(* IEC 61131-3 sources: teller/JD_Teller_LC2_V11/Class/Box_Editer (part 2) *)

            //3-punt 2300
            elsif i = 2 then

                  DoosData^.MinMax[i].T_Max := 2000;
                  DoosData^.MinMax[i].T_Min := 160;
                  DoosData^.MinMax[i].U_Max := 300;
                  DoosData^.MinMax[i].U_Min := 50;
                  DoosData^.MinMax[i].V_Max := 300;
                  DoosData^.MinMax[i].V_Min := 50;
                  DoosData^.MinMax[i].W_Max := 2300;
                  DoosData^.MinMax[i].W_Min := 510;
                  DoosData^.MinMax[i].X_Max := 820;
                  DoosData^.MinMax[i].X_Min := 50;
                  DoosData^.MinMax[i].Y_Max := 820;
                  DoosData^.MinMax[i].Y_Min := 150;
                  DoosData^.MinMax[i].Z_Max := 300;
                  DoosData^.MinMax[i].Z_Min := 0;
                  DoosData^.MinMax[i].Offset_Max := 1150;
                  DoosData^.MinMax[i].Offset_Min := 0;

            //3-punt vakverdeling 2300
            elsif i = 3 then

                  DoosData^.MinMax[i].T_Max := 2000;
                  DoosData^.MinMax[i].T_Min := 320;
                  DoosData^.MinMax[i].U_Max := 300;
                  DoosData^.MinMax[i].U_Min := 30;
                  DoosData^.MinMax[i].V_Max := 300;
                  DoosData^.MinMax[i].V_Min := 30;
                  DoosData^.MinMax[i].W_Max := 1900;
                  DoosData^.MinMax[i].W_Min := 500;
                  DoosData^.MinMax[i].X_Max := 820;
                  DoosData^.MinMax[i].X_Min := 150;
                  DoosData^.MinMax[i].Y_Max := 820;
                  DoosData^.MinMax[i].Y_Min := 100;
                  DoosData^.MinMax[i].Z_Max := 300;
                  DoosData^.MinMax[i].Z_Min := 0;
                  DoosData^.MinMax[i].Offset_Max := 1150;
                  DoosData^.MinMax[i].Offset_Min := 0;

            //4-punt infold 2300
            elsif i = 4 then

                  DoosData^.MinMax[i].T_Max := 2000;
                  DoosData^.MinMax[i].T_Min := 150;
                  DoosData^.MinMax[i].U_Max := 300;
                  DoosData^.MinMax[i].U_Min := 30;
                  DoosData^.MinMax[i].V_Max := 300;
                  DoosData^.MinMax[i].V_Min := 30;
                  DoosData^.MinMax[i].W_Max := 0;
                  DoosData^.MinMax[i].W_Min := 0;
                  DoosData^.MinMax[i].X_Max := 300;
                  DoosData^.MinMax[i].X_Min := 30;
                  DoosData^.MinMax[i].Y_Max := 1480;
                  DoosData^.MinMax[i].Y_Min := 250;
                  DoosData^.MinMax[i].Z_Max := 300;
                  DoosData^.MinMax[i].Z_Min := 0;
                  DoosData^.MinMax[i].Offset_Max := 1150;
                  DoosData^.MinMax[i].Offset_Min := 0;

            //4-punt outfold 2300
            elsif i = 5 then

                  DoosData^.MinMax[i].T_Max := 2000;
                  DoosData^.MinMax[i].T_Min := 150;
                  DoosData^.MinMax[i].U_Max := 300;
                  DoosData^.MinMax[i].U_Min := 30;
                  DoosData^.MinMax[i].V_Max := 300;
                  DoosData^.MinMax[i].V_Min := 30;
                  DoosData^.MinMax[i].W_Max := 0;
                  DoosData^.MinMax[i].W_Min := 0;
                  DoosData^.MinMax[i].X_Max := 300;
                  DoosData^.MinMax[i].X_Min := 30;
                  DoosData^.MinMax[i].Y_Max := 1180;
                  DoosData^.MinMax[i].Y_Min := 250;
                  DoosData^.MinMax[i].Z_Max := 300;
                  DoosData^.MinMax[i].Z_Min := 0;
                  DoosData^.MinMax[i].Offset_Max := 1150;
                  DoosData^.MinMax[i].Offset_Min := 0;

            //4-punt met deksel 2300
            elsif i = 6 then

                  DoosData^.MinMax[i].T_Max := 2000;
                  DoosData^.MinMax[i].T_Min := 150;
                  DoosData^.MinMax[i].U_Max := 300;
                  DoosData^.MinMax[i].U_Min := 30;
                  DoosData^.MinMax[i].V_Max := 300;
                  DoosData^.MinMax[i].V_Min := 30;
                  DoosData^.MinMax[i].W_Max := 2170;
                  DoosData^.MinMax[i].W_Min := 0;
                  DoosData^.MinMax[i].X_Max := 300;
                  DoosData^.MinMax[i].X_Min := 30;
                  DoosData^.MinMax[i].Y_Max := 1480;
                  DoosData^.MinMax[i].Y_Min := 250;
                  DoosData^.MinMax[i].Z_Max := 300;
                  DoosData^.MinMax[i].Z_Min := 0;
                  DoosData^.MinMax[i].Offset_Max := 1150;
                  DoosData^.MinMax[i].Offset_Min := 0;

            //4-punt dubbele wand 2300
            elsif i = 7 then

                  DoosData^.MinMax[i].T_Max := 2000;
                  DoosData^.MinMax[i].T_Min := 150;
                  DoosData^.MinMax[i].U_Max := 300;
                  DoosData^.MinMax[i].U_Min := 30;
                  DoosData^.MinMax[i].V_Max := 300;
                  DoosData^.MinMax[i].V_Min := 30;
                  DoosData^.MinMax[i].W_Max := 2170;
                  DoosData^.MinMax[i].W_Min := 0;
                  DoosData^.MinMax[i].X_Max := 300;
                  DoosData^.MinMax[i].X_Min := 30;
                  DoosData^.MinMax[i].Y_Max := 1480;
                  DoosData^.MinMax[i].Y_Min := 250;
                  DoosData^.MinMax[i].Z_Max := 300;
                  DoosData^.MinMax[i].Z_Min := 0;
                  DoosData^.MinMax[i].Offset_Max := 1150;
                  DoosData^.MinMax[i].Offset_Min := 0;

            //6-punt in/in 2300
            elsif i = 8 then

                  DoosData^.MinMax[i].T_Max := 2000;
                  DoosData^.MinMax[i].T_Min := 150;
                  DoosData^.MinMax[i].U_Max := 300;
                  DoosData^.MinMax[i].U_Min := 30;
                  DoosData^.MinMax[i].V_Max := 300;
                  DoosData^.MinMax[i].V_Min := 30;
                  DoosData^.MinMax[i].W_Max := 2170;
                  DoosData^.MinMax[i].W_Min := 0;
                  DoosData^.MinMax[i].X_Max := 300;
                  DoosData^.MinMax[i].X_Min := 30;
                  DoosData^.MinMax[i].Y_Max := 1480;
                  DoosData^.MinMax[i].Y_Min := 250;
                  DoosData^.MinMax[i].Z_Max := 300;
                  DoosData^.MinMax[i].Z_Min := 0;
                  DoosData^.MinMax[i].Offset_Max := 1150;
                  DoosData^.MinMax[i].Offset_Min := 0;

            //6-punt in/out 2300
            elsif i = 9 then

                  DoosData^.MinMax[i].T_Max := 2000;
                  DoosData^.MinMax[i].T_Min := 150;
                  DoosData^.MinMax[i].U_Max := 300;
                  DoosData^.MinMax[i].U_Min := 30;
                  DoosData^.MinMax[i].V_Max := 300;
                  DoosData^.MinMax[i].V_Min := 30;
                  DoosData^.MinMax[i].W_Max := 2170;
                  DoosData^.MinMax[i].W_Min := 0;
                  DoosData^.MinMax[i].X_Max := 300;
                  DoosData^.MinMax[i].X_Min := 30;
                  DoosData^.MinMax[i].Y_Max := 1480;
                  DoosData^.MinMax[i].Y_Min := 250;
                  DoosData^.MinMax[i].Z_Max := 300;
                  DoosData^.MinMax[i].Z_Min := 0;
                  DoosData^.MinMax[i].Offset_Max := 1150;
                  DoosData^.MinMax[i].Offset_Min := 0;

            //6-punt in/in 2300
            elsif i = 10 then

                  DoosData^.MinMax[i].T_Max := 2000;
                  DoosData^.MinMax[i].T_Min := 150;
                  DoosData^.MinMax[i].U_Max := 300;
                  DoosData^.MinMax[i].U_Min := 30;
                  DoosData^.MinMax[i].V_Max := 300;
                  DoosData^.MinMax[i].V_Min := 30;
                  DoosData^.MinMax[i].W_Max := 2170;
                  DoosData^.MinMax[i].W_Min := 0;
                  DoosData^.MinMax[i].X_Max := 300;
                  DoosData^.MinMax[i].X_Min := 30;
                  DoosData^.MinMax[i].Y_Max := 1480;
                  DoosData^.MinMax[i].Y_Min := 250;
                  DoosData^.MinMax[i].Z_Max := 300;
                  DoosData^.MinMax[i].Z_Min := 0;
                  DoosData^.MinMax[i].Offset_Max := 1150;
                  DoosData^.MinMax[i].Offset_Min := 0;

            //3-punt (gespiegeld) 2300
            elsif i = 11 then

                  DoosData^.MinMax[i].T_Max := 2000;
                  DoosData^.MinMax[i].T_Min := 160;
                  DoosData^.MinMax[i].U_Max := 300;
                  DoosData^.MinMax[i].U_Min := 50;
                  DoosData^.MinMax[i].V_Max := 300;
                  DoosData^.MinMax[i].V_Min := 50;
                  DoosData^.MinMax[i].W_Max := 2300;
                  DoosData^.MinMax[i].W_Min := 510;
                  DoosData^.MinMax[i].X_Max := 820;
                  DoosData^.MinMax[i].X_Min := 50;
                  DoosData^.MinMax[i].Y_Max := 820;
                  DoosData^.MinMax[i].Y_Min := 150;
                  DoosData^.MinMax[i].Z_Max := 300;
                  DoosData^.MinMax[i].Z_Min := 0;
                  DoosData^.MinMax[i].Offset_Max := 1150;
                  DoosData^.MinMax[i].Offset_Min := 0;

            //3-punt (Storaenzo Jonkoping) 2300
            elsif i = 12 then

                  DoosData^.MinMax[i].T_Max := 2000;
                  DoosData^.MinMax[i].T_Min := 160;
                  DoosData^.MinMax[i].U_Max := 300;
                  DoosData^.MinMax[i].U_Min := 50;
                  DoosData^.MinMax[i].V_Max := 300;
                  DoosData^.MinMax[i].V_Min := 50;
                  DoosData^.MinMax[i].W_Max := 2300;
                  DoosData^.MinMax[i].W_Min := 510;
                  DoosData^.MinMax[i].X_Max := 820;
                  DoosData^.MinMax[i].X_Min := 50;
                  DoosData^.MinMax[i].Y_Max := 820;
                  DoosData^.MinMax[i].Y_Min := 150;
                  DoosData^.MinMax[i].Z_Max := 300;
                  DoosData^.MinMax[i].Z_Min := 0;
                  DoosData^.MinMax[i].Offset_Max := 1150;
                  DoosData^.MinMax[i].Offset_Min := 0;

            //langsnaad2 2300
            elsif i = 13 then

                  DoosData^.MinMax[i].T_Max := 2000;
                  DoosData^.MinMax[i].T_Min := 160;
                  DoosData^.MinMax[i].U_Max := 300;
                  DoosData^.MinMax[i].U_Min := 50;
                  DoosData^.MinMax[i].V_Max := 300;
                  DoosData^.MinMax[i].V_Min := 50;
                  DoosData^.MinMax[i].W_Max := 2300;
                  DoosData^.MinMax[i].W_Min := 510;
                  DoosData^.MinMax[i].X_Max := 820;
                  DoosData^.MinMax[i].X_Min := 50;
                  DoosData^.MinMax[i].Y_Max := 820;
                  DoosData^.MinMax[i].Y_Min := 150;
                  DoosData^.MinMax[i].Z_Max := 300;
                  DoosData^.MinMax[i].Z_Min := 0;
                  DoosData^.MinMax[i].Offset_Max := 1150;
                  DoosData^.MinMax[i].Offset_Min := 0;

            //3-punt2 2300
            elsif i = 14 then

                  DoosData^.MinMax[i].T_Max := 2000;
                  DoosData^.MinMax[i].T_Min := 160;
                  DoosData^.MinMax[i].U_Max := 300;
                  DoosData^.MinMax[i].U_Min := 50;
                  DoosData^.MinMax[i].V_Max := 300;
                  DoosData^.MinMax[i].V_Min := 50;
                  DoosData^.MinMax[i].W_Max := 2300;
                  DoosData^.MinMax[i].W_Min := 510;
                  DoosData^.MinMax[i].X_Max := 820;
                  DoosData^.MinMax[i].X_Min := 50;
                  DoosData^.MinMax[i].Y_Max := 820;
                  DoosData^.MinMax[i].Y_Min := 150;
                  DoosData^.MinMax[i].Z_Max := 300;
                  DoosData^.MinMax[i].Z_Min := 0;
                  DoosData^.MinMax[i].Offset_Max := 1150;
                  DoosData^.MinMax[i].Offset_Min := 0;
          end_if;
        end_for;
  end_if;

  if    Presets_MinMax =  m2800 then

        for i:= 1 to 14 do

            DoosData^.MinMax[i].Max_Invoer_Lengte  := 2000;
            DoosData^.MinMax[i].Max_Invoer_Breedte := 2800;

              //langsnaad 2800
            if    i = 1 then

                  DoosData^.MinMax[i].T_Max := 2000;
                  DoosData^.MinMax[i].T_Min := 160;
                  DoosData^.MinMax[i].U_Max := 300;
                  DoosData^.MinMax[i].U_Min := 80;
                  DoosData^.MinMax[i].V_Max := 0;
                  DoosData^.MinMax[i].V_Min := 0;
                  DoosData^.MinMax[i].W_Max := 2800;
                  DoosData^.MinMax[i].W_Min := 510;
                  DoosData^.MinMax[i].X_Max := 1000;
                  DoosData^.MinMax[i].X_Min := 80;
                  DoosData^.MinMax[i].Y_Max := 1000;
                  DoosData^.MinMax[i].Y_Min := 150;
                  DoosData^.MinMax[i].Z_Max := 300;
                  DoosData^.MinMax[i].Z_Min := 0;
                  DoosData^.MinMax[i].Offset_Max := 1400;
                  DoosData^.MinMax[i].Offset_Min := 0;

            //3-punt 2800
            elsif i = 2 then

                  DoosData^.MinMax[i].T_Max := 2000;
                  DoosData^.MinMax[i].T_Min := 160;
                  DoosData^.MinMax[i].U_Max := 300;
                  DoosData^.MinMax[i].U_Min := 80;
                  DoosData^.MinMax[i].V_Max := 300;
                  DoosData^.MinMax[i].V_Min := 80;
                  DoosData^.MinMax[i].W_Max := 2800;
                  DoosData^.MinMax[i].W_Min := 510;
                  DoosData^.MinMax[i].X_Max := 1000;
                  DoosData^.MinMax[i].X_Min := 80;
                  DoosData^.MinMax[i].Y_Max := 1000;
                  DoosData^.MinMax[i].Y_Min := 150;
                  DoosData^.MinMax[i].Z_Max := 300;
                  DoosData^.MinMax[i].Z_Min := 0;
                  DoosData^.MinMax[i].Offset_Max := 1400;
                  DoosData^.MinMax[i].Offset_Min := 0;

            //3-punt vakverdeling 2800
            elsif i = 3 then

                  DoosData^.MinMax[i].T_Max := 2000;
                  DoosData^.MinMax[i].T_Min := 320;
                  DoosData^.MinMax[i].U_Max := 300;
                  DoosData^.MinMax[i].U_Min := 30;
                  DoosData^.MinMax[i].V_Max := 300;
                  DoosData^.MinMax[i].V_Min := 30;
                  DoosData^.MinMax[i].W_Max := 2400;
                  DoosData^.MinMax[i].W_Min := 500;
                  DoosData^.MinMax[i].X_Max := 1000;
                  DoosData^.MinMax[i].X_Min := 150;
                  DoosData^.MinMax[i].Y_Max := 1000;
                  DoosData^.MinMax[i].Y_Min := 100;
                  DoosData^.MinMax[i].Z_Max := 300;
                  DoosData^.MinMax[i].Z_Min := 0;
                  DoosData^.MinMax[i].Offset_Max := 1150;
                  DoosData^.MinMax[i].Offset_Min := 0;

            //4-punt infold 2800
            elsif i = 4 then

                  DoosData^.MinMax[i].T_Max := 2000;
                  DoosData^.MinMax[i].T_Min := 150;
                  DoosData^.MinMax[i].U_Max := 300;
                  DoosData^.MinMax[i].U_Min := 30;
                  DoosData^.MinMax[i].V_Max := 300;
                  DoosData^.MinMax[i].V_Min := 30;
                  DoosData^.MinMax[i].W_Max := 0;
                  DoosData^.MinMax[i].W_Min := 0;
                  DoosData^.MinMax[i].X_Max := 300;
                  DoosData^.MinMax[i].X_Min := 30;
                  DoosData^.MinMax[i].Y_Max := 1480;
                  DoosData^.MinMax[i].Y_Min := 250;
                  DoosData^.MinMax[i].Z_Max := 300;
                  DoosData^.MinMax[i].Z_Min := 0;
                  DoosData^.MinMax[i].Offset_Max := 1150;
                  DoosData^.MinMax[i].Offset_Min := 0;

            //4-punt outfold 2800
            elsif i = 5 then

                  DoosData^.MinMax[i].T_Max := 2000;
                  DoosData^.MinMax[i].T_Min := 150;
                  DoosData^.MinMax[i].U_Max := 300;
                  DoosData^.MinMax[i].U_Min := 30;
                  DoosData^.MinMax[i].V_Max := 300;
                  DoosData^.MinMax[i].V_Min := 30;
                  DoosData^.MinMax[i].W_Max := 0;
                  DoosData^.MinMax[i].W_Min := 0;
                  DoosData^.MinMax[i].X_Max := 300;
                  DoosData^.MinMax[i].X_Min := 30;
                  DoosData^.MinMax[i].Y_Max := 1480;
                  DoosData^.MinMax[i].Y_Min := 250;
                  DoosData^.MinMax[i].Z_Max := 300;
                  DoosData^.MinMax[i].Z_Min := 0;
                  DoosData^.MinMax[i].Offset_Max := 1400;
                  DoosData^.MinMax[i].Offset_Min := 0;

            //4-punt met deksel 2800
            elsif i = 6 then

                  DoosData^.MinMax[i].T_Max := 2000;
                  DoosData^.MinMax[i].T_Min := 150;
                  DoosData^.MinMax[i].U_Max := 300;
                  DoosData^.MinMax[i].U_Min := 30;
                  DoosData^.MinMax[i].V_Max := 300;
                  DoosData^.MinMax[i].V_Min := 30;
                  DoosData^.MinMax[i].W_Max := 2670;
                  DoosData^.MinMax[i].W_Min := 0;
                  DoosData^.MinMax[i].X_Max := 300;
                  DoosData^.MinMax[i].X_Min := 30;
                  DoosData^.MinMax[i].Y_Max := 1480;
                  DoosData^.MinMax[i].Y_Min := 250;
                  DoosData^.MinMax[i].Z_Max := 300;
                  DoosData^.MinMax[i].Z_Min := 0;
                  DoosData^.MinMax[i].Offset_Max := 1150;
                  DoosData^.MinMax[i].Offset_Min := 0;

            //4-punt dubbele wand 2800
            elsif i = 7 then

                  DoosData^.MinMax[i].T_Max := 2000;
                  DoosData^.MinMax[i].T_Min := 150;
                  DoosData^.MinMax[i].U_Max := 300;
                  DoosData^.MinMax[i].U_Min := 30;
                  DoosData^.MinMax[i].V_Max := 300;
                  DoosData^.MinMax[i].V_Min := 30;
                  DoosData^.MinMax[i].W_Max := 2670;
                  DoosData^.MinMax[i].W_Min := 0;
                  DoosData^.MinMax[i].X_Max := 300;
                  DoosData^.MinMax[i].X_Min := 30;
                  DoosData^.MinMax[i].Y_Max := 1480;
                  DoosData^.MinMax[i].Y_Min := 250;
                  DoosData^.MinMax[i].Z_Max := 300;
                  DoosData^.MinMax[i].Z_Min := 0;
                  DoosData^.MinMax[i].Offset_Max := 1150;
                  DoosData^.MinMax[i].Offset_Min := 0;

            //6-punt in/in 2800
            elsif i = 8 then

                  DoosData^.MinMax[i].T_Max := 2000;
                  DoosData^.MinMax[i].T_Min := 150;
                  DoosData^.MinMax[i].U_Max := 300;
                  DoosData^.MinMax[i].U_Min := 30;
                  DoosData^.MinMax[i].V_Max := 300;
                  DoosData^.MinMax[i].V_Min := 30;
                  DoosData^.MinMax[i].W_Max := 2670;
                  DoosData^.MinMax[i].W_Min := 0;
                  DoosData^.MinMax[i].X_Max := 300;
                  DoosData^.MinMax[i].X_Min := 30;
                  DoosData^.MinMax[i].Y_Max := 1480;
                  DoosData^.MinMax[i].Y_Min := 250;
                  DoosData^.MinMax[i].Z_Max := 300;
                  DoosData^.MinMax[i].Z_Min := 0;
                  DoosData^.MinMax[i].Offset_Max := 1150;
                  DoosData^.MinMax[i].Offset_Min := 0;

            //6-punt in/out 2800
            elsif i = 9 then

                  DoosData^.MinMax[i].T_Max := 2000;
                  DoosData^.MinMax[i].T_Min := 150;
                  DoosData^.MinMax[i].U_Max := 300;
                  DoosData^.MinMax[i].U_Min := 30;
                  DoosData^.MinMax[i].V_Max := 300;
                  DoosData^.MinMax[i].V_Min := 30;
                  DoosData^.MinMax[i].W_Max := 2670;
                  DoosData^.MinMax[i].W_Min := 0;
                  DoosData^.MinMax[i].X_Max := 300;
                  DoosData^.MinMax[i].X_Min := 30;
                  DoosData^.MinMax[i].Y_Max := 1480;
                  DoosData^.MinMax[i].Y_Min := 250;
                  DoosData^.MinMax[i].Z_Max := 300;
                  DoosData^.MinMax[i].Z_Min := 0;
                  DoosData^.MinMax[i].Offset_Max := 1150;
                  DoosData^.MinMax[i].Offset_Min := 0;

            //6-punt in/in 2800
            elsif i = 10 then

                  DoosData^.MinMax[i].T_Max := 2000;
                  DoosData^.MinMax[i].T_Min := 150;
                  DoosData^.MinMax[i].U_Max := 300;
                  DoosData^.MinMax[i].U_Min := 30;
                  DoosData^.MinMax[i].V_Max := 300;
                  DoosData^.MinMax[i].V_Min := 30;
                  DoosData^.MinMax[i].W_Max := 2670;
                  DoosData^.MinMax[i].W_Min := 0;
                  DoosData^.MinMax[i].X_Max := 300;
                  DoosData^.MinMax[i].X_Min := 30;
                  DoosData^.MinMax[i].Y_Max := 1480;
                  DoosData^.MinMax[i].Y_Min := 250;
                  DoosData^.MinMax[i].Z_Max := 300;
                  DoosData^.MinMax[i].Z_Min := 0;
                  DoosData^.MinMax[i].Offset_Max := 1150;
                  DoosData^.MinMax[i].Offset_Min := 0;

            //3-punt (gespiegeld) 2800
            elsif i = 11 then

                  DoosData^.MinMax[i].T_Max := 2000;
                  DoosData^.MinMax[i].T_Min := 160;
                  DoosData^.MinMax[i].U_Max := 300;
                  DoosData^.MinMax[i].U_Min := 80;
                  DoosData^.MinMax[i].V_Max := 300;
                  DoosData^.MinMax[i].V_Min := 80;
                  DoosData^.MinMax[i].W_Max := 2800;
                  DoosData^.MinMax[i].W_Min := 510;
                  DoosData^.MinMax[i].X_Max := 1000;
                  DoosData^.MinMax[i].X_Min := 80;
                  DoosData^.MinMax[i].Y_Max := 1000;
                  DoosData^.MinMax[i].Y_Min := 150;
                  DoosData^.MinMax[i].Z_Max := 300;
                  DoosData^.MinMax[i].Z_Min := 0;
                  DoosData^.MinMax[i].Offset_Max := 1400;
                  DoosData^.MinMax[i].Offset_Min := 0;

            //3-punt (Storaenzo Jonkoping) 2800
            elsif i = 12 then

                  DoosData^.MinMax[i].T_Max := 2000;
                  DoosData^.MinMax[i].T_Min := 160;
                  DoosData^.MinMax[i].U_Max := 300;
                  DoosData^.MinMax[i].U_Min := 80;
                  DoosData^.MinMax[i].V_Max := 300;
                  DoosData^.MinMax[i].V_Min := 80;
                  DoosData^.MinMax[i].W_Max := 2800;
                  DoosData^.MinMax[i].W_Min := 510;
                  DoosData^.MinMax[i].X_Max := 1000;
                  DoosData^.MinMax[i].X_Min := 80;
                  DoosData^.MinMax[i].Y_Max := 1000;
                  DoosData^.MinMax[i].Y_Min := 150;
                  DoosData^.MinMax[i].Z_Max := 300;
                  DoosData^.MinMax[i].Z_Min := 0;
                  DoosData^.MinMax[i].Offset_Max := 1400;
                  DoosData^.MinMax[i].Offset_Min := 0;

            //langsnaad2 2800
            elsif i = 13 then

                  DoosData^.MinMax[i].T_Max := 2000;
                  DoosData^.MinMax[i].T_Min := 160;
                  DoosData^.MinMax[i].U_Max := 300;
                  DoosData^.MinMax[i].U_Min := 80;
                  DoosData^.MinMax[i].V_Max := 300;
                  DoosData^.MinMax[i].V_Min := 80;
                  DoosData^.MinMax[i].W_Max := 2800;
                  DoosData^.MinMax[i].W_Min := 510;
                  DoosData^.MinMax[i].X_Max := 1000;
                  DoosData^.MinMax[i].X_Min := 80;
                  DoosData^.MinMax[i].Y_Max := 1000;
                  DoosData^.MinMax[i].Y_Min := 150;
                  DoosData^.MinMax[i].Z_Max := 300;
                  DoosData^.MinMax[i].Z_Min := 0;
                  DoosData^.MinMax[i].Offset_Max := 1400;
                  DoosData^.MinMax[i].Offset_Min := 0;

            //3-punt2 2800
            elsif i = 14 then

                  DoosData^.MinMax[i].T_Max := 2000;
                  DoosData^.MinMax[i].T_Min := 160;
                  DoosData^.MinMax[i].U_Max := 300;
                  DoosData^.MinMax[i].U_Min := 80;
                  DoosData^.MinMax[i].V_Max := 300;
                  DoosData^.MinMax[i].V_Min := 80;
                  DoosData^.MinMax[i].W_Max := 2800;
                  DoosData^.MinMax[i].W_Min := 510;
                  DoosData^.MinMax[i].X_Max := 1000;
                  DoosData^.MinMax[i].X_Min := 80;
                  DoosData^.MinMax[i].Y_Max := 1000;
                  DoosData^.MinMax[i].Y_Min := 150;
                  DoosData^.MinMax[i].Z_Max := 300;
                  DoosData^.MinMax[i].Z_Min := 0;
                  DoosData^.MinMax[i].Offset_Max := 1400;
                  DoosData^.MinMax[i].Offset_Min := 0;
            end_if;
        end_for;
  end_if;

  c_Refresh_Values01.Write (c_Refresh_Values01);
  c_Refresh_Values02.Write (c_Refresh_Values02);
  c_Refresh_Values03.Write (c_Refresh_Values03);
  c_Refresh_Values04.Write (c_Refresh_Values04);
  c_Refresh_Values05.Write (c_Refresh_Values05);
  c_Refresh_Values06.Write (c_Refresh_Values06);
  c_Refresh_Values07.Write (c_Refresh_Values07);
  c_Refresh_Values08.Write (c_Refresh_Values08);
  c_Refresh_Values09.Write (c_Refresh_Values09);
  c_Refresh_Values10.Write (c_Refresh_Values10);
  c_Refresh_Values11.Write (c_Refresh_Values11);
  c_Refresh_Values12.Write (c_Refresh_Values12);
  c_Refresh_Values13.Write (c_Refresh_Values13);
  c_Refresh_Values14.Write (c_Refresh_Values14);

 	result := Presets_MinMax;

END_FUNCTION

FUNCTION VIRTUAL GLOBAL Box_Editer::ResetValues::Write
	VAR_INPUT
		input (EAX) 	: DINT;
	END_VAR
	VAR_OUTPUT
		result (EAX) 	: DINT;
	END_VAR

	ResetValues := input;

  //Reset van de doosparameters

  s_T := 0;
  s_U := 0;
  s_V := 0;
  s_W := 0;
  s_X := 0;
  s_Y := 0;
  s_Z := 0;

 	result := ResetValues;

END_FUNCTION
